// SIMATIC S7-200 SMART project (STEP 7-Micro/WIN SMART), CPU ST20

SYMBOL_TABLE System Symbols
Always_On        SM0.0    // Always ON
First_Scan_On    SM0.1    // ON for the first scan cycle only
END_SYMBOL_TABLE

ORGANIZATION_BLOCK MAIN:OB1
TITLE=Modbus RTU Multi-point Digital Controller RKC MA900/MA901
BEGIN
Network 1
// Network Comment
LD     Always_On:SM0.0
=      L60.0
LD     Always_On:SM0.0
=      L63.7
LD     L60.0
CALL   MBUS_CTRL:SBR1, L63.7, 19200, 0, 0, 250, M0.0, VB10
Network 2
LD     First_Scan_On:SM0.1
S      M8.0, 1
Network 3
LD     M8.0
O      M8.1
TON    T98, 10
Network 4
LD     T98
EU
S      M1.0, 1
R      M8.0, 2
Network 5
// Measured value (PV)
LD     M1.0
=      L60.0
LD     M1.0
EU
=      L63.7
LD     L60.0
CALL   MBUS_MSG:SBR2, L63.7, 1, 0, 40001, +8, &VB100, M0.1, VB11
Network 6
LD     M1.0
S      M1.1, 1
R      M1.0, 1
Network 7
// Set value (SV)
LD     M1.1
=      L60.0
LD     M1.1
EU
=      L63.7
LD     L60.0
CALL   MBUS_MSG:SBR2, L63.7, 1, 1, 40201, +8, &VB120, M0.2, VB12
Network 8
LD     M0.2
S      M1.2, 1
R      M1.1, 1
Network 9
// Used / unused of channels
LD     M1.2
=      L60.0
LD     M1.2
EU
=      L63.7
LD     L60.0
CALL   MBUS_MSG:SBR2, L63.7, 1, 1, 40441, +8, &VB154, M0.3, VB13
Network 10
LD     M0.3
S      M1.3, 1
R      M1.2, 1
Network 11
// Manipulated output value
LD     M1.3
=      L60.0
LD     M1.3
EU
=      L63.7
LD     L60.0
CALL   MBUS_MSG:SBR2, L63.7, 1, 0, 40021, +8, &VB180, M0.4, VB14
Network 12
LD     M0.4
R      M1.3, 1
EU
S      M8.1, 1
END_ORGANIZATION_BLOCK

// SBR1: protected block, not included

// SBR2: protected block, not included

// SBR3: protected block, not included
